// TIA Portal V20 export
FUNCTION "FIT101" : Void   // FC19, FBD
{ S7_Optimized_Access := 'TRUE' }
// stored: SetENOAutomatically false
   VAR_TEMP
      Temp : "DigVal";
      Temp_1 : "DigVal";
   END_VAR
BEGIN

REGION Network 1: Channel input
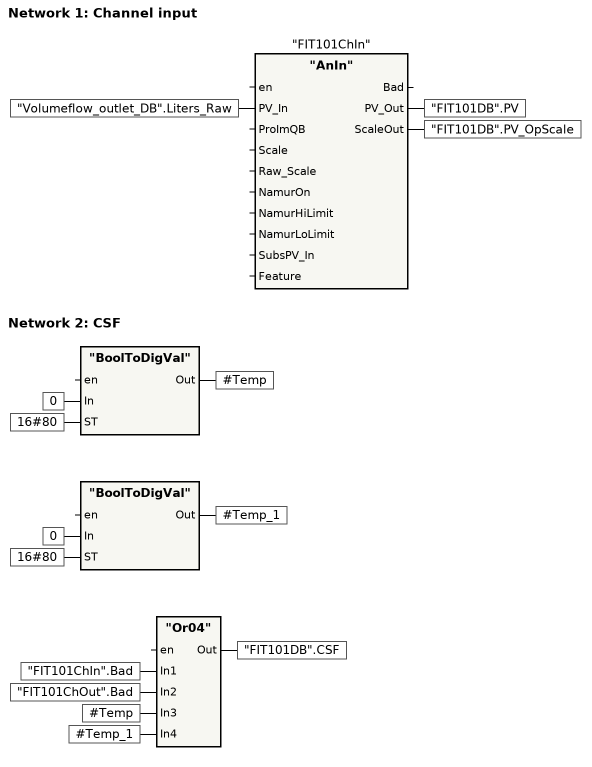
   "FIT101ChIn"(PV_In := "Volumeflow_outlet_DB".Liters_Raw,   // "AnIn"
                PV_Out => "FIT101DB".PV,
                ScaleOut => "FIT101DB".PV_OpScale);
END_REGION

REGION Network 2: CSF
   "BoolToDigVal"(In := 0, ST := 16#80, Out => #Temp);
   "BoolToDigVal"(In := 0, ST := 16#80, Out => #Temp_1);
   "Or04"(In1 := "FIT101ChIn".Bad,
          In2 := "FIT101ChOut".Bad,
          In3 := #Temp,
          In4 := #Temp_1,
          Out => "FIT101DB".CSF);
END_REGION

REGION Network 3: MonAnL
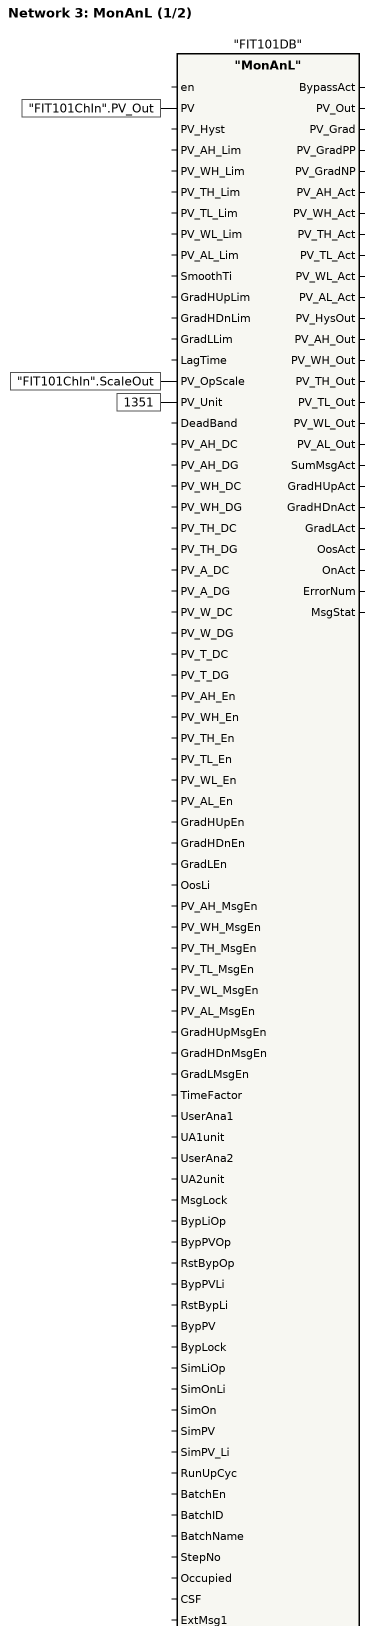
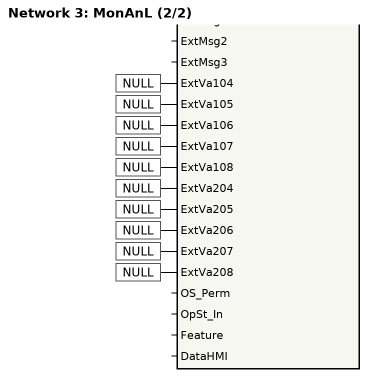
   "FIT101DB"(PV := "FIT101ChIn".PV_Out,   // "MonAnL"
              PV_OpScale := "FIT101ChIn".ScaleOut,
              PV_Unit := 1351,
              ExtVa104 := NULL,
              ExtVa105 := NULL,
              ExtVa106 := NULL,
              ExtVa107 := NULL,
              ExtVa108 := NULL,
              ExtVa204 := NULL,
              ExtVa205 := NULL,
              ExtVa206 := NULL,
              ExtVa207 := NULL,
              ExtVa208 := NULL);
END_REGION

REGION Network 4: MTP
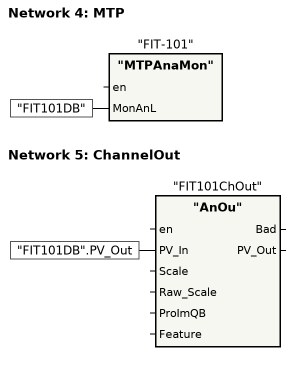
   "FIT-101"(MonAnL := "FIT101DB");   // "MTPAnaMon"
END_REGION

REGION Network 5: ChannelOut
   "FIT101ChOut"(PV_In := "FIT101DB".PV_Out);   // "AnOu"
END_REGION
END_FUNCTION
